TYPE Angles :
STRUCT
	theta1_right	:LREAL;
	theta2_left		:LREAL;
END_STRUCT
END_TYPE

(* stored: Version 1.1.0.1, ProductVersion 3.1.4024.13
   DUT Angles: Id {9d894569-ab16-4cb0-99a1-a071639ffc4d} *)
